// TIA Portal V20 export
TYPE "LER_typePDR"
// stored: Access Published
   STRUCT
      parent_Tracecode : Array[1..20] of Char;
      parent_PartNumber : Array[1..8] of Char;
      child_Tracecode : Array[1..20] of Char;
   END_STRUCT;
END_TYPE
